Staubli VAL3: PA_grinding_V3.dtx

public tool tTool = {z=100, fatherId=flange[0], ioLink=valve1}
public frame fWork = {fatherId=world[0]}
public jointRx j_home = {j1=83.61, j2=38.15, j3=96.24, j4=-4.09, j5=-58.18, j6=-4.12}
public jointRx j_scan = {j1=83.61, j2=38.15, j3=96.24, j4=-4.09, j5=-58.18, j6=-4.12}
public jointRx jWaypoints[100]
public num nWaypointCount
public num nForceTarget
public num nDOC
public num nCmdSignal
public num nStatusSignal
num nLastCmd
bool bRunning
num i
mdesc mNomSpeed = {tmax=200, rmax=200, blend=off}
mdesc mGrindSpeed = {tmax=30, rmax=30, leave=1, reach=1, blend=off}
public sio siTcpIpCommand = {link=Socket\Command}
public sio siTcpIpMotion = {link=Socket\Motion}
public sio siTcpIpFbk = {link=Socket\Feedback}
public num nConnFlag
num nByte
public pointRx curent_pos = {fatherId=world[0]}
mdesc mAprSpeed = {tmax=5, rmax=5, blend=off}
public aio aiECAT1_0 = {link=EtherCAT-1\%IF0}
public aio aoECAT1_0 = {link=EtherCAT-1\%QF0}
public aio aoECAT1_32 = {link=EtherCAT-1\%QF32}
public aio aoECAT1_64 = {link=EtherCAT-1\%QF64}
public aio aoECAT1_96 = {link=EtherCAT-1\%QF96}
public aio aoECAT1_128 = {link=EtherCAT-1\%QF128}
public aio aoECAT1_160 = {link=EtherCAT-1\%QF160}
